{attribute 'qualified_only'}
{attribute 'strict'}
{attribute 'to_string'}
TYPE eUgridPowerMode :
(
	auto 			:= 0,
	DroopZeroStart	:= 1,
	Droop			:= 2,
	Isochronous		:= 3,
	None			:= 4
);
END_TYPE

(* stored: Version 1.1.0.1, ProductVersion 3.1.4026.18
   DUT eUgridPowerMode: Id {ac2e2075-032b-4d23-82bb-5ecd17f4a6bf} *)
